FUNCTION_BLOCK FB_AxisEnable
VAR_INPUT
END_VAR
VAR_OUTPUT
END_VAR
VAR
	fbXAxis: MC_Power;
	fbYAxis: MC_Power;
	fbZAxis: MC_Power;
END_VAR

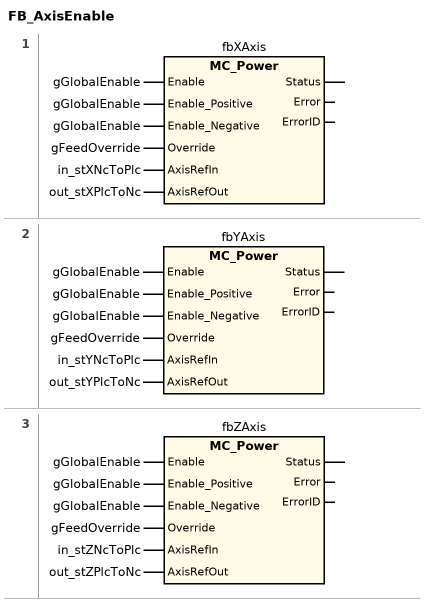
// NETWORK 1
fbXAxis(
    Enable := gGlobalEnable,
    Enable_Positive := gGlobalEnable,
    Enable_Negative := gGlobalEnable,
    Override := gFeedOverride,
    AxisRefIn := in_stXNcToPlc,
    AxisRefOut := out_stXPlcToNc); // MC_Power

// NETWORK 2
fbYAxis(
    Enable := gGlobalEnable,
    Enable_Positive := gGlobalEnable,
    Enable_Negative := gGlobalEnable,
    Override := gFeedOverride,
    AxisRefIn := in_stYNcToPlc,
    AxisRefOut := out_stYPlcToNc); // MC_Power

// NETWORK 3
fbZAxis(
    Enable := gGlobalEnable,
    Enable_Positive := gGlobalEnable,
    Enable_Negative := gGlobalEnable,
    Override := gFeedOverride,
    AxisRefIn := in_stZNcToPlc,
    AxisRefOut := out_stZPlcToNc); // MC_Power

END_FUNCTION_BLOCK

(* stored: Version 1.1.0.1, ProductVersion 3.1.4024.10
   POU FB_AxisEnable: Id {2e285c4e-74ca-4757-802c-1b0b592a9546}, SpecialFunc None *)
